FUNCTION_BLOCK SkillFB (* Composite FB wrapping other FBs *)
  (* Standard: 61499-2 *)
  (* Version 1.0, 2021-03-18, AK120569 *)
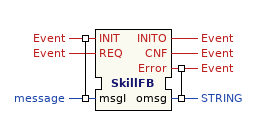
  EVENT_INPUT
    INIT WITH msgI; (* Initialization Request *)
    REQ; (* Normal Execution Request *)
  END_EVENT
  EVENT_OUTPUT
    INITO; (* Initialization Confirm *)
    CNF; (* Execution Confirmation *)
    Error WITH omsg;
  END_EVENT
  VAR_INPUT
    msgI : message;
  END_VAR
  VAR_OUTPUT
    omsg : STRING;
  END_VAR
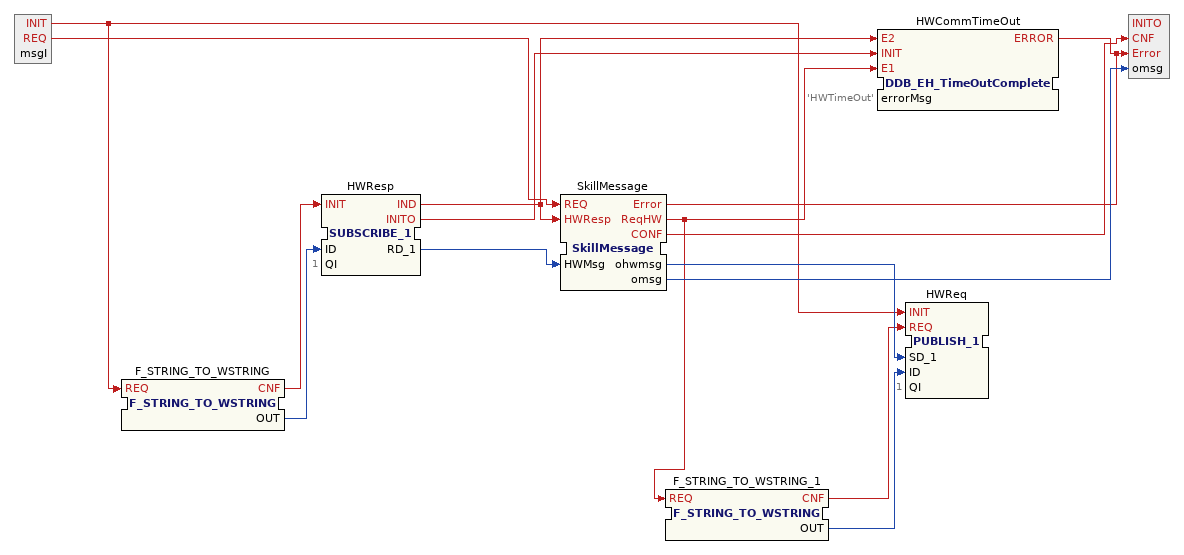
  FBS
    HWReq : PUBLISH_1(QI := 1);
    HWResp : SUBSCRIBE_1(QI := 1);
    HWCommTimeOut : DDB_EH_TimeOutComplete(errorMsg := 'HWTimeOut');
    SkillMessage : SkillMessage;
    F_STRING_TO_WSTRING : F_STRING_TO_WSTRING;
    F_STRING_TO_WSTRING_1 : F_STRING_TO_WSTRING;
  END_FBS
  EVENT_CONNECTIONS
    INIT TO HWReq.INIT;
    HWCommTimeOut.ERROR TO Error;
    HWResp.IND TO HWCommTimeOut.E2;
    HWResp.INITO TO HWCommTimeOut.INIT;
    REQ TO SkillMessage.REQ;
    HWResp.IND TO SkillMessage.HWResp;
    SkillMessage.Error TO Error;
    SkillMessage.ReqHW TO HWCommTimeOut.E1;
    SkillMessage.CONF TO CNF;
    INIT TO F_STRING_TO_WSTRING.REQ;
    F_STRING_TO_WSTRING.CNF TO HWResp.INIT;
    SkillMessage.ReqHW TO F_STRING_TO_WSTRING_1.REQ;
    F_STRING_TO_WSTRING_1.CNF TO HWReq.REQ;
  END_CONNECTIONS
  DATA_CONNECTIONS
    HWResp.RD_1 TO SkillMessage.HWMsg;
    SkillMessage.ohwmsg TO HWReq.SD_1;
    SkillMessage.omsg TO omsg;
    F_STRING_TO_WSTRING.OUT TO HWResp.ID;
    F_STRING_TO_WSTRING_1.OUT TO HWReq.ID;
  END_CONNECTIONS
END_FUNCTION_BLOCK
